// TIA Portal V17 export
// export: Created 2025-03-05T08:03:12.6134683Z, ExportSetting WithDefaults, DisplayName Totally Integrated Automation Portal, DisplayVersion V17 Update 8, DisplayName TIA Portal Openness, DisplayVersion V17 Update 8, DisplayName TIA Portal Version Control Interface, DisplayVersion V17, DisplayName SINAMICS Startdrive Advanced, DisplayVersion V17 SP2, DisplayName SINAMICS Startdrive G110M, G120, G120C, G120D, G120P, G115D, DisplayVersion V17 SP2, DisplayName SINAMICS Startdrive G130, G150, S120, S150, SINAMICS MV, S210, DisplayVersion V17 SP2, DisplayName STEP 7 Professional, DisplayVersion V17 Update 8, DisplayName SINUMERIK ONE STEP 7 Toolbox, DisplayVersion V17 Update 12, DisplayName SINUMERIK 840D sl STEP 7 Toolbox, DisplayVersion V17 Update 12, DisplayName STEP 7 Safety, DisplayVersion V17 Update 6, DisplayName WinCC Advanced, DisplayVersion V17 Update 8
FUNCTION "FC22500_HOPPER_SYSTEM_CONTROLS" : Void   // FC22500, LAD
TITLE = FC22500 HOPPER SYSTEM CONTROLS
{ S7_Optimized_Access := 'TRUE' }
VERSION : 0.1
// stored: AutoNumber false, IsIECCheckEnabled false, SetENOAutomatically false, UDAEnableTagReadback false
   VAR_TEMP
      RPM_INT_AUX : Word;
      RPM_REAL_AUX : Real;
   END_VAR
BEGIN

REGION Network 1: //////////UNIT 01 HOPERS CONTROLS//////////
END_REGION

REGION Network 2: CALL FB22501 TEMPERATURE JKT CONTROL UPPER HOPPER 1 UNIT 01
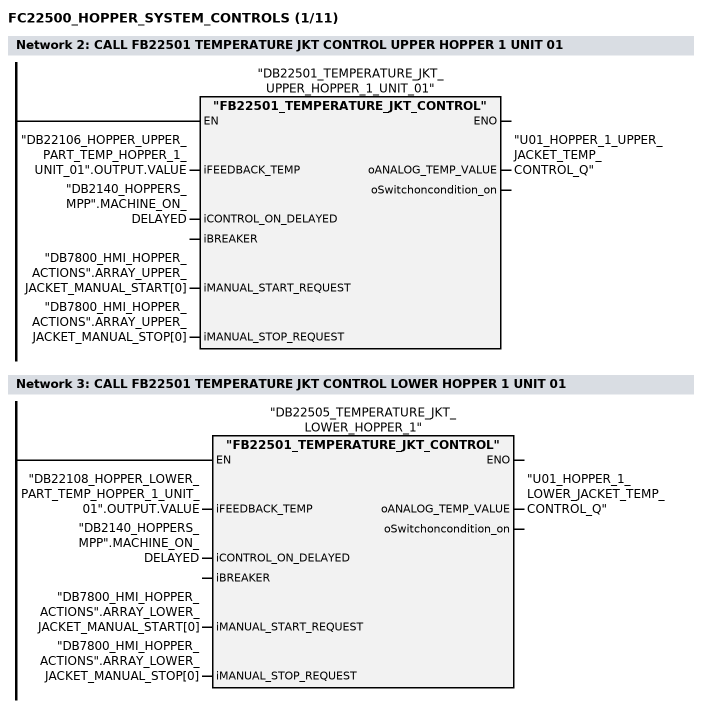
   RUNG wire#powerrail
      "DB22501_TEMPERATURE_JKT_UPPER_HOPPER_1_UNIT_01"(iFEEDBACK_TEMP := "DB22106_HOPPER_UPPER_PART_TEMP_HOPPER_1_UNIT_01".OUTPUT.VALUE, iCONTROL_ON_DELAYED := "DB2140_HOPPERS_MPP".MACHINE_ON_DELAYED, iBREAKER :=, iMANUAL_START_REQUEST := "DB7800_HMI_HOPPER_ACTIONS".ARRAY_UPPER_JACKET_MANUAL_START[0], iMANUAL_STOP_REQUEST := "DB7800_HMI_HOPPER_ACTIONS".ARRAY_UPPER_JACKET_MANUAL_STOP[0], oANALOG_TEMP_VALUE => "U01_HOPPER_1_UPPER_JACKET_TEMP_CONTROL_Q", oSwitchoncondition_on =>)
   END_RUNG
   // the same network as SCL:
   "DB22501_TEMPERATURE_JKT_UPPER_HOPPER_1_UNIT_01"(iFEEDBACK_TEMP := "DB22106_HOPPER_UPPER_PART_TEMP_HOPPER_1_UNIT_01".OUTPUT.VALUE,   // "FB22501_TEMPERATURE_JKT_CONTROL"
                           iCONTROL_ON_DELAYED := "DB2140_HOPPERS_MPP".MACHINE_ON_DELAYED,
                           iMANUAL_START_REQUEST := "DB7800_HMI_HOPPER_ACTIONS".ARRAY_UPPER_JACKET_MANUAL_START[0],
                           iMANUAL_STOP_REQUEST := "DB7800_HMI_HOPPER_ACTIONS".ARRAY_UPPER_JACKET_MANUAL_STOP[0],
                           oANALOG_TEMP_VALUE => "U01_HOPPER_1_UPPER_JACKET_TEMP_CONTROL_Q");
END_REGION

REGION Network 3: CALL FB22501 TEMPERATURE JKT CONTROL LOWER HOPPER 1 UNIT 01
   RUNG wire#powerrail
      "DB22505_TEMPERATURE_JKT_LOWER_HOPPER_1"(iFEEDBACK_TEMP := "DB22108_HOPPER_LOWER_PART_TEMP_HOPPER_1_UNIT_01".OUTPUT.VALUE, iCONTROL_ON_DELAYED := "DB2140_HOPPERS_MPP".MACHINE_ON_DELAYED, iBREAKER :=, iMANUAL_START_REQUEST := "DB7800_HMI_HOPPER_ACTIONS".ARRAY_LOWER_JACKET_MANUAL_START[0], iMANUAL_STOP_REQUEST := "DB7800_HMI_HOPPER_ACTIONS".ARRAY_LOWER_JACKET_MANUAL_STOP[0], oANALOG_TEMP_VALUE => "U01_HOPPER_1_LOWER_JACKET_TEMP_CONTROL_Q", oSwitchoncondition_on =>)
   END_RUNG
   // the same network as SCL:
   "DB22505_TEMPERATURE_JKT_LOWER_HOPPER_1"(iFEEDBACK_TEMP := "DB22108_HOPPER_LOWER_PART_TEMP_HOPPER_1_UNIT_01".OUTPUT.VALUE,   // "FB22501_TEMPERATURE_JKT_CONTROL"
                           iCONTROL_ON_DELAYED := "DB2140_HOPPERS_MPP".MACHINE_ON_DELAYED,
                           iMANUAL_START_REQUEST := "DB7800_HMI_HOPPER_ACTIONS".ARRAY_LOWER_JACKET_MANUAL_START[0],
                           iMANUAL_STOP_REQUEST := "DB7800_HMI_HOPPER_ACTIONS".ARRAY_LOWER_JACKET_MANUAL_STOP[0],
                           oANALOG_TEMP_VALUE => "U01_HOPPER_1_LOWER_JACKET_TEMP_CONTROL_Q");
END_REGION

REGION Network 4: CALL FB22502 MOTOR STIRRER CONTROL HOPPER 1 UNIT 01
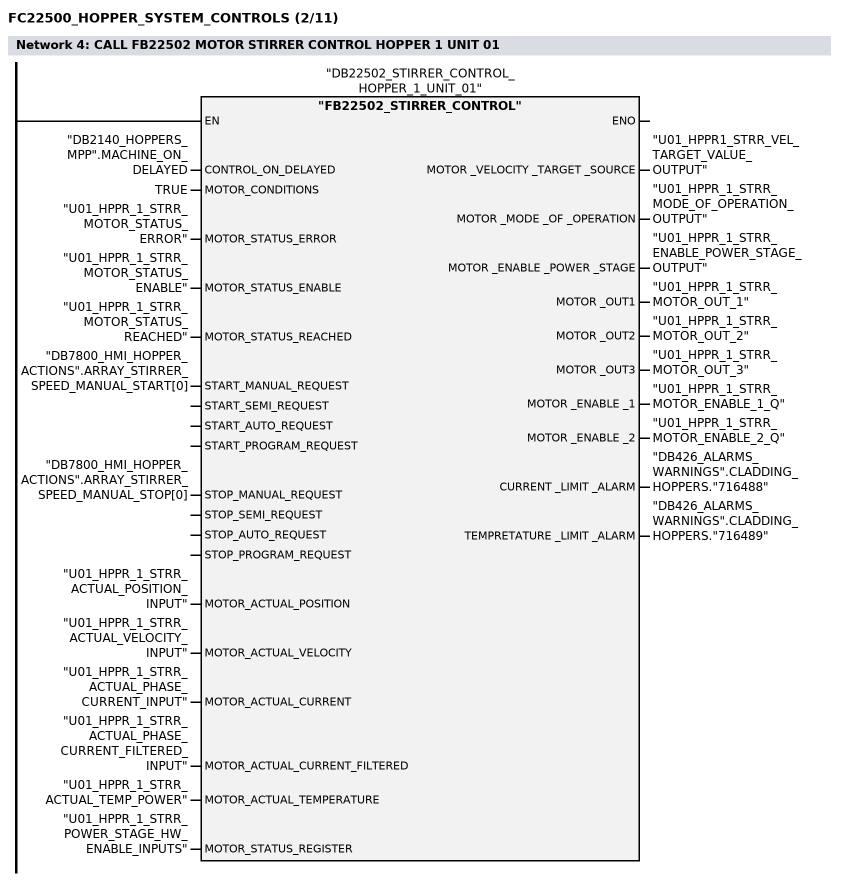
   RUNG wire#powerrail
      "DB22502_STIRRER_CONTROL_HOPPER_1_UNIT_01"(CONTROL_ON_DELAYED := "DB2140_HOPPERS_MPP".MACHINE_ON_DELAYED, MOTOR_CONDITIONS := TRUE, MOTOR_STATUS_ERROR := "U01_HPPR_1_STRR_MOTOR_STATUS_ERROR", MOTOR_STATUS_ENABLE := "U01_HPPR_1_STRR_MOTOR_STATUS_ENABLE", MOTOR_STATUS_REACHED := "U01_HPPR_1_STRR_MOTOR_STATUS_REACHED", START_MANUAL_REQUEST := "DB7800_HMI_HOPPER_ACTIONS".ARRAY_STIRRER_SPEED_MANUAL_START[0], START_SEMI_REQUEST :=, START_AUTO_REQUEST :=, START_PROGRAM_REQUEST :=, STOP_MANUAL_REQUEST := "DB7800_HMI_HOPPER_ACTIONS".ARRAY_STIRRER_SPEED_MANUAL_STOP[0], STOP_SEMI_REQUEST :=, STOP_AUTO_REQUEST :=, STOP_PROGRAM_REQUEST :=, MOTOR_ACTUAL_POSITION := "U01_HPPR_1_STRR_ACTUAL_POSITION_INPUT", MOTOR_ACTUAL_VELOCITY := "U01_HPPR_1_STRR_ACTUAL_VELOCITY_INPUT", MOTOR_ACTUAL_CURRENT := "U01_HPPR_1_STRR_ACTUAL_PHASE_CURRENT_INPUT", MOTOR_ACTUAL_CURRENT_FILTERED := "U01_HPPR_1_STRR_ACTUAL_PHASE_CURRENT_FILTERED_INPUT", MOTOR_ACTUAL_TEMPERATURE := "U01_HPPR_1_STRR_ACTUAL_TEMP_POWER", MOTOR_STATUS_REGISTER := "U01_HPPR_1_STRR_POWER_STAGE_HW_ENABLE_INPUTS", "MOTOR _VELOCITY _TARGET _SOURCE" => "U01_HPPR1_STRR_VEL_TARGET_VALUE_OUTPUT", "MOTOR _MODE _OF _OPERATION" => "U01_HPPR_1_STRR_MODE_OF_OPERATION_OUTPUT", "MOTOR _ENABLE _POWER _STAGE" => "U01_HPPR_1_STRR_ENABLE_POWER_STAGE_OUTPUT", "MOTOR _OUT1" => "U01_HPPR_1_STRR_MOTOR_OUT_1", "MOTOR _OUT2" => "U01_HPPR_1_STRR_MOTOR_OUT_2", "MOTOR _OUT3" => "U01_HPPR_1_STRR_MOTOR_OUT_3", "MOTOR _ENABLE _1" => "U01_HPPR_1_STRR_MOTOR_ENABLE_1_Q", "MOTOR _ENABLE _2" => "U01_HPPR_1_STRR_MOTOR_ENABLE_2_Q", "CURRENT _LIMIT _ALARM" => "DB426_ALARMS_WARNINGS".CLADDING_HOPPERS."716488", "TEMPRETATURE _LIMIT _ALARM" => "DB426_ALARMS_WARNINGS".CLADDING_HOPPERS."716489")
   END_RUNG
   // the same network as SCL:
   "DB22502_STIRRER_CONTROL_HOPPER_1_UNIT_01"(CONTROL_ON_DELAYED := "DB2140_HOPPERS_MPP".MACHINE_ON_DELAYED,   // "FB22502_STIRRER_CONTROL"
                           MOTOR_CONDITIONS := TRUE,
                           MOTOR_STATUS_ERROR := "U01_HPPR_1_STRR_MOTOR_STATUS_ERROR",
                           MOTOR_STATUS_ENABLE := "U01_HPPR_1_STRR_MOTOR_STATUS_ENABLE",
                           MOTOR_STATUS_REACHED := "U01_HPPR_1_STRR_MOTOR_STATUS_REACHED",
                           START_MANUAL_REQUEST := "DB7800_HMI_HOPPER_ACTIONS".ARRAY_STIRRER_SPEED_MANUAL_START[0],
                           STOP_MANUAL_REQUEST := "DB7800_HMI_HOPPER_ACTIONS".ARRAY_STIRRER_SPEED_MANUAL_STOP[0],
                           MOTOR_ACTUAL_POSITION := "U01_HPPR_1_STRR_ACTUAL_POSITION_INPUT",
                           MOTOR_ACTUAL_VELOCITY := "U01_HPPR_1_STRR_ACTUAL_VELOCITY_INPUT",
                           MOTOR_ACTUAL_CURRENT := "U01_HPPR_1_STRR_ACTUAL_PHASE_CURRENT_INPUT",
                           MOTOR_ACTUAL_CURRENT_FILTERED := "U01_HPPR_1_STRR_ACTUAL_PHASE_CURRENT_FILTERED_INPUT",
                           MOTOR_ACTUAL_TEMPERATURE := "U01_HPPR_1_STRR_ACTUAL_TEMP_POWER",
                           MOTOR_STATUS_REGISTER := "U01_HPPR_1_STRR_POWER_STAGE_HW_ENABLE_INPUTS",
                           "MOTOR _VELOCITY _TARGET _SOURCE" => "U01_HPPR1_STRR_VEL_TARGET_VALUE_OUTPUT",
                           "MOTOR _MODE _OF _OPERATION" => "U01_HPPR_1_STRR_MODE_OF_OPERATION_OUTPUT",
                           "MOTOR _ENABLE _POWER _STAGE" => "U01_HPPR_1_STRR_ENABLE_POWER_STAGE_OUTPUT",
                           "MOTOR _OUT1" => "U01_HPPR_1_STRR_MOTOR_OUT_1",
                           "MOTOR _OUT2" => "U01_HPPR_1_STRR_MOTOR_OUT_2",
                           "MOTOR _OUT3" => "U01_HPPR_1_STRR_MOTOR_OUT_3",
                           "MOTOR _ENABLE _1" => "U01_HPPR_1_STRR_MOTOR_ENABLE_1_Q",
                           "MOTOR _ENABLE _2" => "U01_HPPR_1_STRR_MOTOR_ENABLE_2_Q",
                           "CURRENT _LIMIT _ALARM" => "DB426_ALARMS_WARNINGS".CLADDING_HOPPERS."716488",
                           "TEMPRETATURE _LIMIT _ALARM" => "DB426_ALARMS_WARNINGS".CLADDING_HOPPERS."716489");
END_REGION

REGION Network 5: CALL FB22503 HOPPER COVER PRESSURE CONTROL HOPPER 1 UNIT 01
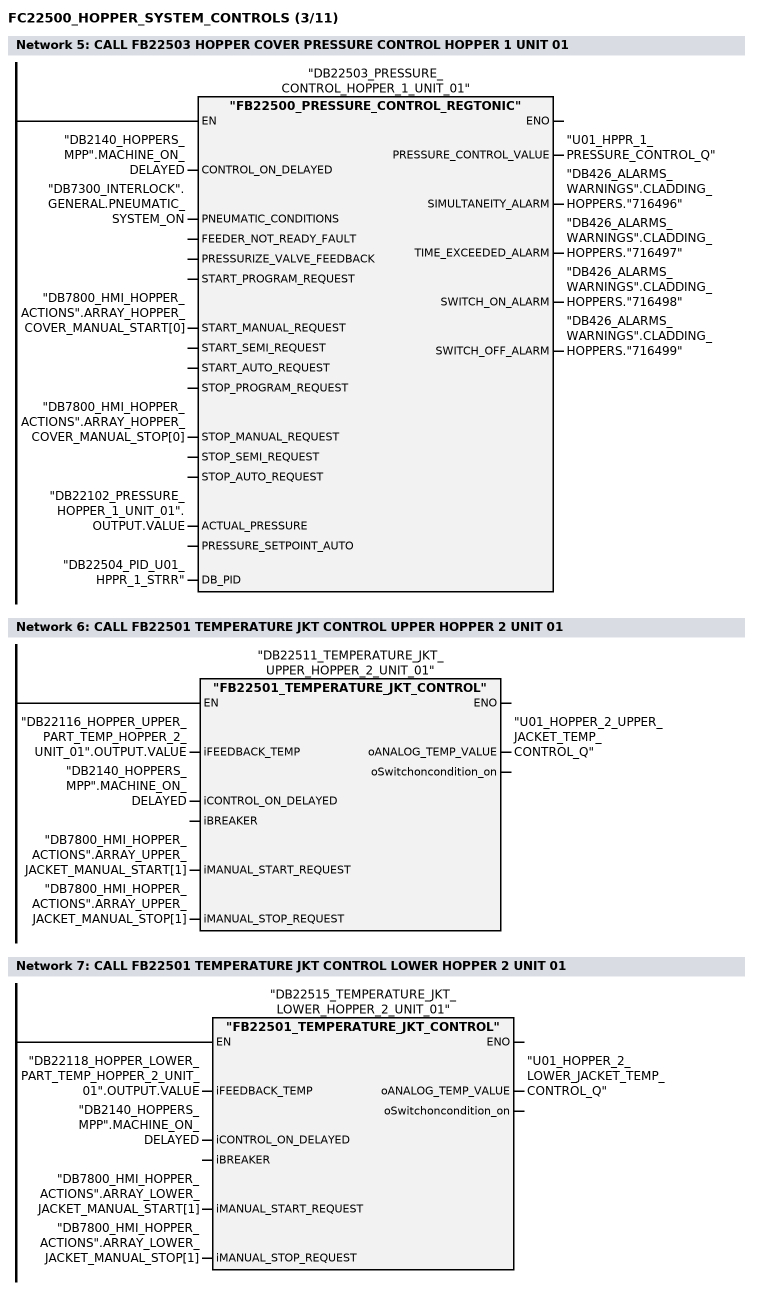
   RUNG wire#powerrail
      "DB22503_PRESSURE_CONTROL_HOPPER_1_UNIT_01"(CONTROL_ON_DELAYED := "DB2140_HOPPERS_MPP".MACHINE_ON_DELAYED, PNEUMATIC_CONDITIONS := "DB7300_INTERLOCK".GENERAL.PNEUMATIC_SYSTEM_ON, FEEDER_NOT_READY_FAULT :=, PRESSURIZE_VALVE_FEEDBACK :=, START_PROGRAM_REQUEST :=, START_MANUAL_REQUEST := "DB7800_HMI_HOPPER_ACTIONS".ARRAY_HOPPER_COVER_MANUAL_START[0], START_SEMI_REQUEST :=, START_AUTO_REQUEST :=, STOP_PROGRAM_REQUEST :=, STOP_MANUAL_REQUEST := "DB7800_HMI_HOPPER_ACTIONS".ARRAY_HOPPER_COVER_MANUAL_STOP[0], STOP_SEMI_REQUEST :=, STOP_AUTO_REQUEST :=, ACTUAL_PRESSURE := "DB22102_PRESSURE_HOPPER_1_UNIT_01".OUTPUT.VALUE, PRESSURE_SETPOINT_AUTO :=, DB_PID := "DB22504_PID_U01_HPPR_1_STRR", PRESSURE_CONTROL_VALUE => "U01_HPPR_1_PRESSURE_CONTROL_Q", SIMULTANEITY_ALARM => "DB426_ALARMS_WARNINGS".CLADDING_HOPPERS."716496", TIME_EXCEEDED_ALARM => "DB426_ALARMS_WARNINGS".CLADDING_HOPPERS."716497", SWITCH_ON_ALARM => "DB426_ALARMS_WARNINGS".CLADDING_HOPPERS."716498", SWITCH_OFF_ALARM => "DB426_ALARMS_WARNINGS".CLADDING_HOPPERS."716499")
   END_RUNG
   // the same network as SCL:
   "DB22503_PRESSURE_CONTROL_HOPPER_1_UNIT_01"(CONTROL_ON_DELAYED := "DB2140_HOPPERS_MPP".MACHINE_ON_DELAYED,   // "FB22500_PRESSURE_CONTROL_REGTONIC"
                           PNEUMATIC_CONDITIONS := "DB7300_INTERLOCK".GENERAL.PNEUMATIC_SYSTEM_ON,
                           START_MANUAL_REQUEST := "DB7800_HMI_HOPPER_ACTIONS".ARRAY_HOPPER_COVER_MANUAL_START[0],
                           STOP_MANUAL_REQUEST := "DB7800_HMI_HOPPER_ACTIONS".ARRAY_HOPPER_COVER_MANUAL_STOP[0],
                           ACTUAL_PRESSURE := "DB22102_PRESSURE_HOPPER_1_UNIT_01".OUTPUT.VALUE,
                           DB_PID := "DB22504_PID_U01_HPPR_1_STRR",
                           PRESSURE_CONTROL_VALUE => "U01_HPPR_1_PRESSURE_CONTROL_Q",
                           SIMULTANEITY_ALARM => "DB426_ALARMS_WARNINGS".CLADDING_HOPPERS."716496",
                           TIME_EXCEEDED_ALARM => "DB426_ALARMS_WARNINGS".CLADDING_HOPPERS."716497",
                           SWITCH_ON_ALARM => "DB426_ALARMS_WARNINGS".CLADDING_HOPPERS."716498",
                           SWITCH_OFF_ALARM => "DB426_ALARMS_WARNINGS".CLADDING_HOPPERS."716499");
END_REGION

REGION Network 6: CALL FB22501 TEMPERATURE JKT CONTROL UPPER HOPPER 2 UNIT 01
   RUNG wire#powerrail
      "DB22511_TEMPERATURE_JKT_UPPER_HOPPER_2_UNIT_01"(iFEEDBACK_TEMP := "DB22116_HOPPER_UPPER_PART_TEMP_HOPPER_2_UNIT_01".OUTPUT.VALUE, iCONTROL_ON_DELAYED := "DB2140_HOPPERS_MPP".MACHINE_ON_DELAYED, iBREAKER :=, iMANUAL_START_REQUEST := "DB7800_HMI_HOPPER_ACTIONS".ARRAY_UPPER_JACKET_MANUAL_START[1], iMANUAL_STOP_REQUEST := "DB7800_HMI_HOPPER_ACTIONS".ARRAY_UPPER_JACKET_MANUAL_STOP[1], oANALOG_TEMP_VALUE => "U01_HOPPER_2_UPPER_JACKET_TEMP_CONTROL_Q", oSwitchoncondition_on =>)
   END_RUNG
   // the same network as SCL:
   "DB22511_TEMPERATURE_JKT_UPPER_HOPPER_2_UNIT_01"(iFEEDBACK_TEMP := "DB22116_HOPPER_UPPER_PART_TEMP_HOPPER_2_UNIT_01".OUTPUT.VALUE,   // "FB22501_TEMPERATURE_JKT_CONTROL"
                           iCONTROL_ON_DELAYED := "DB2140_HOPPERS_MPP".MACHINE_ON_DELAYED,
                           iMANUAL_START_REQUEST := "DB7800_HMI_HOPPER_ACTIONS".ARRAY_UPPER_JACKET_MANUAL_START[1],
                           iMANUAL_STOP_REQUEST := "DB7800_HMI_HOPPER_ACTIONS".ARRAY_UPPER_JACKET_MANUAL_STOP[1],
                           oANALOG_TEMP_VALUE => "U01_HOPPER_2_UPPER_JACKET_TEMP_CONTROL_Q");
END_REGION

REGION Network 7: CALL FB22501 TEMPERATURE JKT CONTROL LOWER HOPPER 2 UNIT 01
   RUNG wire#powerrail
      "DB22515_TEMPERATURE_JKT_LOWER_HOPPER_2_UNIT_01"(iFEEDBACK_TEMP := "DB22118_HOPPER_LOWER_PART_TEMP_HOPPER_2_UNIT_01".OUTPUT.VALUE, iCONTROL_ON_DELAYED := "DB2140_HOPPERS_MPP".MACHINE_ON_DELAYED, iBREAKER :=, iMANUAL_START_REQUEST := "DB7800_HMI_HOPPER_ACTIONS".ARRAY_LOWER_JACKET_MANUAL_START[1], iMANUAL_STOP_REQUEST := "DB7800_HMI_HOPPER_ACTIONS".ARRAY_LOWER_JACKET_MANUAL_STOP[1], oANALOG_TEMP_VALUE => "U01_HOPPER_2_LOWER_JACKET_TEMP_CONTROL_Q", oSwitchoncondition_on =>)
   END_RUNG
   // the same network as SCL:
   "DB22515_TEMPERATURE_JKT_LOWER_HOPPER_2_UNIT_01"(iFEEDBACK_TEMP := "DB22118_HOPPER_LOWER_PART_TEMP_HOPPER_2_UNIT_01".OUTPUT.VALUE,   // "FB22501_TEMPERATURE_JKT_CONTROL"
                           iCONTROL_ON_DELAYED := "DB2140_HOPPERS_MPP".MACHINE_ON_DELAYED,
                           iMANUAL_START_REQUEST := "DB7800_HMI_HOPPER_ACTIONS".ARRAY_LOWER_JACKET_MANUAL_START[1],
                           iMANUAL_STOP_REQUEST := "DB7800_HMI_HOPPER_ACTIONS".ARRAY_LOWER_JACKET_MANUAL_STOP[1],
                           oANALOG_TEMP_VALUE => "U01_HOPPER_2_LOWER_JACKET_TEMP_CONTROL_Q");
END_REGION

REGION Network 8: CALL FB22502 MOTOR STIRRER CONTROL HOPPER 2 UNIT 01
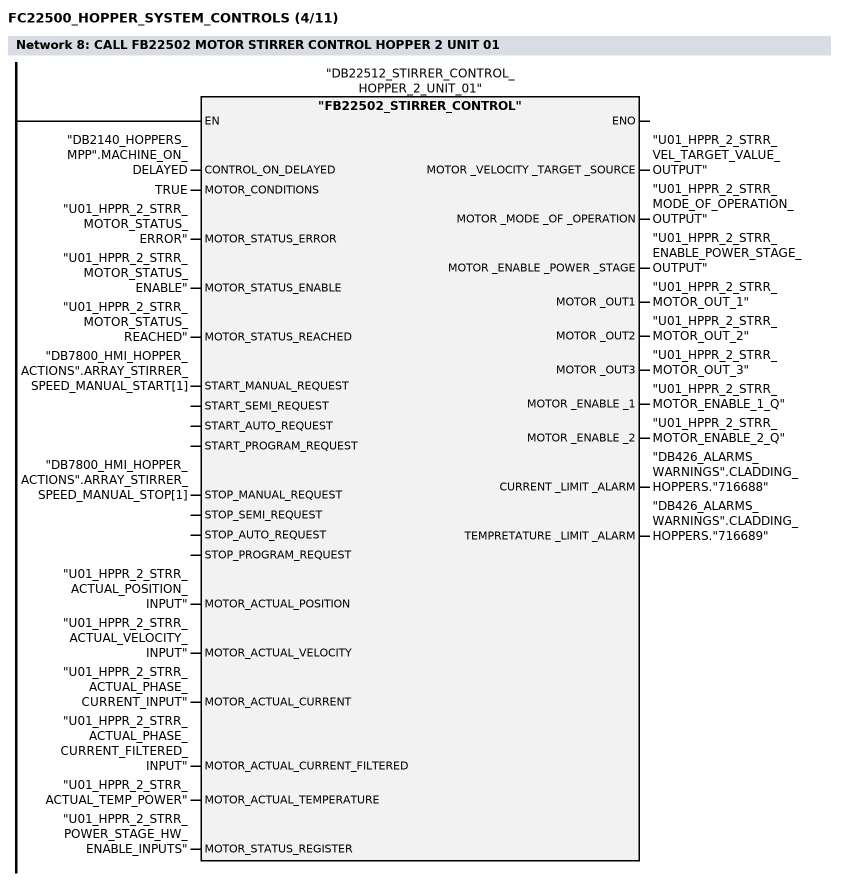
   RUNG wire#powerrail
      "DB22512_STIRRER_CONTROL_HOPPER_2_UNIT_01"(CONTROL_ON_DELAYED := "DB2140_HOPPERS_MPP".MACHINE_ON_DELAYED, MOTOR_CONDITIONS := TRUE, MOTOR_STATUS_ERROR := "U01_HPPR_2_STRR_MOTOR_STATUS_ERROR", MOTOR_STATUS_ENABLE := "U01_HPPR_2_STRR_MOTOR_STATUS_ENABLE", MOTOR_STATUS_REACHED := "U01_HPPR_2_STRR_MOTOR_STATUS_REACHED", START_MANUAL_REQUEST := "DB7800_HMI_HOPPER_ACTIONS".ARRAY_STIRRER_SPEED_MANUAL_START[1], START_SEMI_REQUEST :=, START_AUTO_REQUEST :=, START_PROGRAM_REQUEST :=, STOP_MANUAL_REQUEST := "DB7800_HMI_HOPPER_ACTIONS".ARRAY_STIRRER_SPEED_MANUAL_STOP[1], STOP_SEMI_REQUEST :=, STOP_AUTO_REQUEST :=, STOP_PROGRAM_REQUEST :=, MOTOR_ACTUAL_POSITION := "U01_HPPR_2_STRR_ACTUAL_POSITION_INPUT", MOTOR_ACTUAL_VELOCITY := "U01_HPPR_2_STRR_ACTUAL_VELOCITY_INPUT", MOTOR_ACTUAL_CURRENT := "U01_HPPR_2_STRR_ACTUAL_PHASE_CURRENT_INPUT", MOTOR_ACTUAL_CURRENT_FILTERED := "U01_HPPR_2_STRR_ACTUAL_PHASE_CURRENT_FILTERED_INPUT", MOTOR_ACTUAL_TEMPERATURE := "U01_HPPR_2_STRR_ACTUAL_TEMP_POWER", MOTOR_STATUS_REGISTER := "U01_HPPR_2_STRR_POWER_STAGE_HW_ENABLE_INPUTS", "MOTOR _VELOCITY _TARGET _SOURCE" => "U01_HPPR_2_STRR_VEL_TARGET_VALUE_OUTPUT", "MOTOR _MODE _OF _OPERATION" => "U01_HPPR_2_STRR_MODE_OF_OPERATION_OUTPUT", "MOTOR _ENABLE _POWER _STAGE" => "U01_HPPR_2_STRR_ENABLE_POWER_STAGE_OUTPUT", "MOTOR _OUT1" => "U01_HPPR_2_STRR_MOTOR_OUT_1", "MOTOR _OUT2" => "U01_HPPR_2_STRR_MOTOR_OUT_2", "MOTOR _OUT3" => "U01_HPPR_2_STRR_MOTOR_OUT_3", "MOTOR _ENABLE _1" => "U01_HPPR_2_STRR_MOTOR_ENABLE_1_Q", "MOTOR _ENABLE _2" => "U01_HPPR_2_STRR_MOTOR_ENABLE_2_Q", "CURRENT _LIMIT _ALARM" => "DB426_ALARMS_WARNINGS".CLADDING_HOPPERS."716688", "TEMPRETATURE _LIMIT _ALARM" => "DB426_ALARMS_WARNINGS".CLADDING_HOPPERS."716689")
   END_RUNG
   // the same network as SCL:
   "DB22512_STIRRER_CONTROL_HOPPER_2_UNIT_01"(CONTROL_ON_DELAYED := "DB2140_HOPPERS_MPP".MACHINE_ON_DELAYED,   // "FB22502_STIRRER_CONTROL"
                           MOTOR_CONDITIONS := TRUE,
                           MOTOR_STATUS_ERROR := "U01_HPPR_2_STRR_MOTOR_STATUS_ERROR",
                           MOTOR_STATUS_ENABLE := "U01_HPPR_2_STRR_MOTOR_STATUS_ENABLE",
                           MOTOR_STATUS_REACHED := "U01_HPPR_2_STRR_MOTOR_STATUS_REACHED",
                           START_MANUAL_REQUEST := "DB7800_HMI_HOPPER_ACTIONS".ARRAY_STIRRER_SPEED_MANUAL_START[1],
                           STOP_MANUAL_REQUEST := "DB7800_HMI_HOPPER_ACTIONS".ARRAY_STIRRER_SPEED_MANUAL_STOP[1],
                           MOTOR_ACTUAL_POSITION := "U01_HPPR_2_STRR_ACTUAL_POSITION_INPUT",
                           MOTOR_ACTUAL_VELOCITY := "U01_HPPR_2_STRR_ACTUAL_VELOCITY_INPUT",
                           MOTOR_ACTUAL_CURRENT := "U01_HPPR_2_STRR_ACTUAL_PHASE_CURRENT_INPUT",
                           MOTOR_ACTUAL_CURRENT_FILTERED := "U01_HPPR_2_STRR_ACTUAL_PHASE_CURRENT_FILTERED_INPUT",
                           MOTOR_ACTUAL_TEMPERATURE := "U01_HPPR_2_STRR_ACTUAL_TEMP_POWER",
                           MOTOR_STATUS_REGISTER := "U01_HPPR_2_STRR_POWER_STAGE_HW_ENABLE_INPUTS",
                           "MOTOR _VELOCITY _TARGET _SOURCE" => "U01_HPPR_2_STRR_VEL_TARGET_VALUE_OUTPUT",
                           "MOTOR _MODE _OF _OPERATION" => "U01_HPPR_2_STRR_MODE_OF_OPERATION_OUTPUT",
                           "MOTOR _ENABLE _POWER _STAGE" => "U01_HPPR_2_STRR_ENABLE_POWER_STAGE_OUTPUT",
                           "MOTOR _OUT1" => "U01_HPPR_2_STRR_MOTOR_OUT_1",
                           "MOTOR _OUT2" => "U01_HPPR_2_STRR_MOTOR_OUT_2",
                           "MOTOR _OUT3" => "U01_HPPR_2_STRR_MOTOR_OUT_3",
                           "MOTOR _ENABLE _1" => "U01_HPPR_2_STRR_MOTOR_ENABLE_1_Q",
                           "MOTOR _ENABLE _2" => "U01_HPPR_2_STRR_MOTOR_ENABLE_2_Q",
                           "CURRENT _LIMIT _ALARM" => "DB426_ALARMS_WARNINGS".CLADDING_HOPPERS."716688",
                           "TEMPRETATURE _LIMIT _ALARM" => "DB426_ALARMS_WARNINGS".CLADDING_HOPPERS."716689");
END_REGION

REGION Network 9: CALL FB22503 HOPPER PRESSURE CONTROL HOPPER 2 UNIT 01
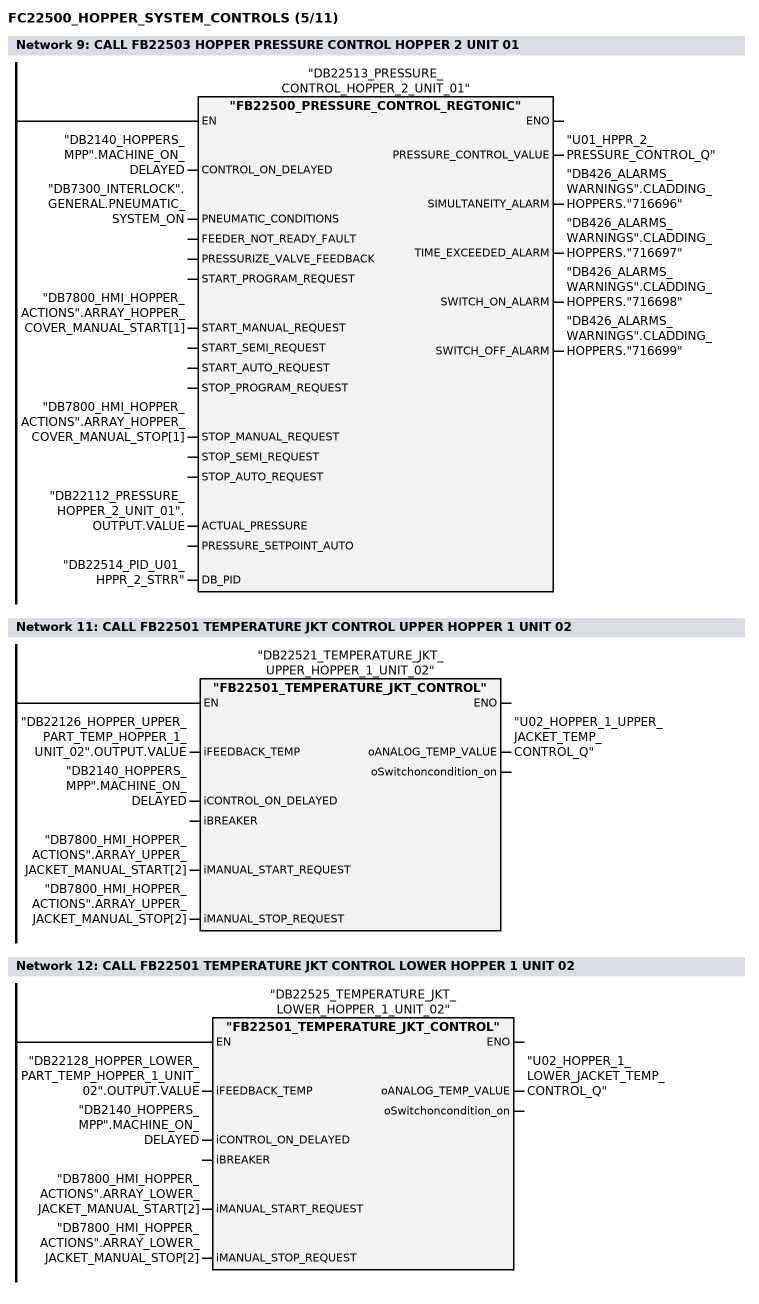
   RUNG wire#powerrail
      "DB22513_PRESSURE_CONTROL_HOPPER_2_UNIT_01"(CONTROL_ON_DELAYED := "DB2140_HOPPERS_MPP".MACHINE_ON_DELAYED, PNEUMATIC_CONDITIONS := "DB7300_INTERLOCK".GENERAL.PNEUMATIC_SYSTEM_ON, FEEDER_NOT_READY_FAULT :=, PRESSURIZE_VALVE_FEEDBACK :=, START_PROGRAM_REQUEST :=, START_MANUAL_REQUEST := "DB7800_HMI_HOPPER_ACTIONS".ARRAY_HOPPER_COVER_MANUAL_START[1], START_SEMI_REQUEST :=, START_AUTO_REQUEST :=, STOP_PROGRAM_REQUEST :=, STOP_MANUAL_REQUEST := "DB7800_HMI_HOPPER_ACTIONS".ARRAY_HOPPER_COVER_MANUAL_STOP[1], STOP_SEMI_REQUEST :=, STOP_AUTO_REQUEST :=, ACTUAL_PRESSURE := "DB22112_PRESSURE_HOPPER_2_UNIT_01".OUTPUT.VALUE, PRESSURE_SETPOINT_AUTO :=, DB_PID := "DB22514_PID_U01_HPPR_2_STRR", PRESSURE_CONTROL_VALUE => "U01_HPPR_2_PRESSURE_CONTROL_Q", SIMULTANEITY_ALARM => "DB426_ALARMS_WARNINGS".CLADDING_HOPPERS."716696", TIME_EXCEEDED_ALARM => "DB426_ALARMS_WARNINGS".CLADDING_HOPPERS."716697", SWITCH_ON_ALARM => "DB426_ALARMS_WARNINGS".CLADDING_HOPPERS."716698", SWITCH_OFF_ALARM => "DB426_ALARMS_WARNINGS".CLADDING_HOPPERS."716699")
   END_RUNG
   // the same network as SCL:
   "DB22513_PRESSURE_CONTROL_HOPPER_2_UNIT_01"(CONTROL_ON_DELAYED := "DB2140_HOPPERS_MPP".MACHINE_ON_DELAYED,   // "FB22500_PRESSURE_CONTROL_REGTONIC"
                           PNEUMATIC_CONDITIONS := "DB7300_INTERLOCK".GENERAL.PNEUMATIC_SYSTEM_ON,
                           START_MANUAL_REQUEST := "DB7800_HMI_HOPPER_ACTIONS".ARRAY_HOPPER_COVER_MANUAL_START[1],
                           STOP_MANUAL_REQUEST := "DB7800_HMI_HOPPER_ACTIONS".ARRAY_HOPPER_COVER_MANUAL_STOP[1],
                           ACTUAL_PRESSURE := "DB22112_PRESSURE_HOPPER_2_UNIT_01".OUTPUT.VALUE,
                           DB_PID := "DB22514_PID_U01_HPPR_2_STRR",
                           PRESSURE_CONTROL_VALUE => "U01_HPPR_2_PRESSURE_CONTROL_Q",
                           SIMULTANEITY_ALARM => "DB426_ALARMS_WARNINGS".CLADDING_HOPPERS."716696",
                           TIME_EXCEEDED_ALARM => "DB426_ALARMS_WARNINGS".CLADDING_HOPPERS."716697",
                           SWITCH_ON_ALARM => "DB426_ALARMS_WARNINGS".CLADDING_HOPPERS."716698",
                           SWITCH_OFF_ALARM => "DB426_ALARMS_WARNINGS".CLADDING_HOPPERS."716699");
END_REGION

REGION Network 10: //////////UNIT 02 HOPERS CONTROLS//////////
END_REGION

REGION Network 11: CALL FB22501 TEMPERATURE JKT CONTROL UPPER HOPPER 1 UNIT 02
   RUNG wire#powerrail
      "DB22521_TEMPERATURE_JKT_UPPER_HOPPER_1_UNIT_02"(iFEEDBACK_TEMP := "DB22126_HOPPER_UPPER_PART_TEMP_HOPPER_1_UNIT_02".OUTPUT.VALUE, iCONTROL_ON_DELAYED := "DB2140_HOPPERS_MPP".MACHINE_ON_DELAYED, iBREAKER :=, iMANUAL_START_REQUEST := "DB7800_HMI_HOPPER_ACTIONS".ARRAY_UPPER_JACKET_MANUAL_START[2], iMANUAL_STOP_REQUEST := "DB7800_HMI_HOPPER_ACTIONS".ARRAY_UPPER_JACKET_MANUAL_STOP[2], oANALOG_TEMP_VALUE => "U02_HOPPER_1_UPPER_JACKET_TEMP_CONTROL_Q", oSwitchoncondition_on =>)
   END_RUNG
   // the same network as SCL:
   "DB22521_TEMPERATURE_JKT_UPPER_HOPPER_1_UNIT_02"(iFEEDBACK_TEMP := "DB22126_HOPPER_UPPER_PART_TEMP_HOPPER_1_UNIT_02".OUTPUT.VALUE,   // "FB22501_TEMPERATURE_JKT_CONTROL"
                           iCONTROL_ON_DELAYED := "DB2140_HOPPERS_MPP".MACHINE_ON_DELAYED,
                           iMANUAL_START_REQUEST := "DB7800_HMI_HOPPER_ACTIONS".ARRAY_UPPER_JACKET_MANUAL_START[2],
                           iMANUAL_STOP_REQUEST := "DB7800_HMI_HOPPER_ACTIONS".ARRAY_UPPER_JACKET_MANUAL_STOP[2],
                           oANALOG_TEMP_VALUE => "U02_HOPPER_1_UPPER_JACKET_TEMP_CONTROL_Q");
END_REGION

REGION Network 12: CALL FB22501 TEMPERATURE JKT CONTROL LOWER HOPPER 1 UNIT 02
   RUNG wire#powerrail
      "DB22525_TEMPERATURE_JKT_LOWER_HOPPER_1_UNIT_02"(iFEEDBACK_TEMP := "DB22128_HOPPER_LOWER_PART_TEMP_HOPPER_1_UNIT_02".OUTPUT.VALUE, iCONTROL_ON_DELAYED := "DB2140_HOPPERS_MPP".MACHINE_ON_DELAYED, iBREAKER :=, iMANUAL_START_REQUEST := "DB7800_HMI_HOPPER_ACTIONS".ARRAY_LOWER_JACKET_MANUAL_START[2], iMANUAL_STOP_REQUEST := "DB7800_HMI_HOPPER_ACTIONS".ARRAY_LOWER_JACKET_MANUAL_STOP[2], oANALOG_TEMP_VALUE => "U02_HOPPER_1_LOWER_JACKET_TEMP_CONTROL_Q", oSwitchoncondition_on =>)
   END_RUNG
   // the same network as SCL:
   "DB22525_TEMPERATURE_JKT_LOWER_HOPPER_1_UNIT_02"(iFEEDBACK_TEMP := "DB22128_HOPPER_LOWER_PART_TEMP_HOPPER_1_UNIT_02".OUTPUT.VALUE,   // "FB22501_TEMPERATURE_JKT_CONTROL"
                           iCONTROL_ON_DELAYED := "DB2140_HOPPERS_MPP".MACHINE_ON_DELAYED,
                           iMANUAL_START_REQUEST := "DB7800_HMI_HOPPER_ACTIONS".ARRAY_LOWER_JACKET_MANUAL_START[2],
                           iMANUAL_STOP_REQUEST := "DB7800_HMI_HOPPER_ACTIONS".ARRAY_LOWER_JACKET_MANUAL_STOP[2],
                           oANALOG_TEMP_VALUE => "U02_HOPPER_1_LOWER_JACKET_TEMP_CONTROL_Q");
END_REGION

REGION Network 13: CALL FB22502 MOTOR STIRRER CONTROL HOPPER 1 UNIT 02
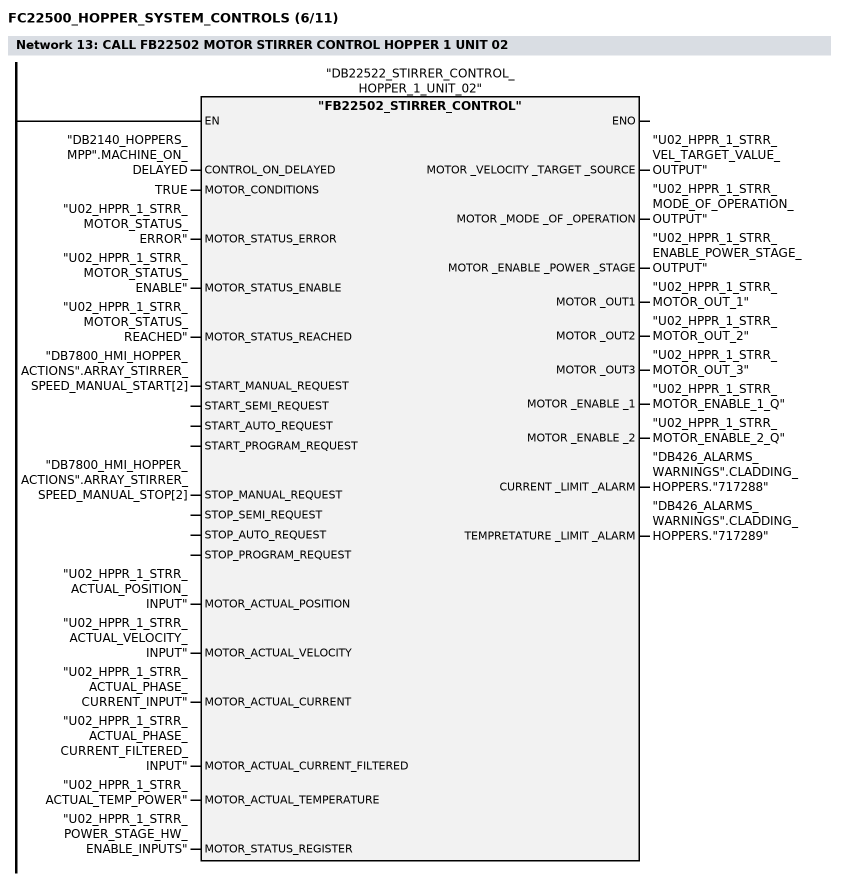
   RUNG wire#powerrail
      "DB22522_STIRRER_CONTROL_HOPPER_1_UNIT_02"(CONTROL_ON_DELAYED := "DB2140_HOPPERS_MPP".MACHINE_ON_DELAYED, MOTOR_CONDITIONS := TRUE, MOTOR_STATUS_ERROR := "U02_HPPR_1_STRR_MOTOR_STATUS_ERROR", MOTOR_STATUS_ENABLE := "U02_HPPR_1_STRR_MOTOR_STATUS_ENABLE", MOTOR_STATUS_REACHED := "U02_HPPR_1_STRR_MOTOR_STATUS_REACHED", START_MANUAL_REQUEST := "DB7800_HMI_HOPPER_ACTIONS".ARRAY_STIRRER_SPEED_MANUAL_START[2], START_SEMI_REQUEST :=, START_AUTO_REQUEST :=, START_PROGRAM_REQUEST :=, STOP_MANUAL_REQUEST := "DB7800_HMI_HOPPER_ACTIONS".ARRAY_STIRRER_SPEED_MANUAL_STOP[2], STOP_SEMI_REQUEST :=, STOP_AUTO_REQUEST :=, STOP_PROGRAM_REQUEST :=, MOTOR_ACTUAL_POSITION := "U02_HPPR_1_STRR_ACTUAL_POSITION_INPUT", MOTOR_ACTUAL_VELOCITY := "U02_HPPR_1_STRR_ACTUAL_VELOCITY_INPUT", MOTOR_ACTUAL_CURRENT := "U02_HPPR_1_STRR_ACTUAL_PHASE_CURRENT_INPUT", MOTOR_ACTUAL_CURRENT_FILTERED := "U02_HPPR_1_STRR_ACTUAL_PHASE_CURRENT_FILTERED_INPUT", MOTOR_ACTUAL_TEMPERATURE := "U02_HPPR_1_STRR_ACTUAL_TEMP_POWER", MOTOR_STATUS_REGISTER := "U02_HPPR_1_STRR_POWER_STAGE_HW_ENABLE_INPUTS", "MOTOR _VELOCITY _TARGET _SOURCE" => "U02_HPPR_1_STRR_VEL_TARGET_VALUE_OUTPUT", "MOTOR _MODE _OF _OPERATION" => "U02_HPPR_1_STRR_MODE_OF_OPERATION_OUTPUT", "MOTOR _ENABLE _POWER _STAGE" => "U02_HPPR_1_STRR_ENABLE_POWER_STAGE_OUTPUT", "MOTOR _OUT1" => "U02_HPPR_1_STRR_MOTOR_OUT_1", "MOTOR _OUT2" => "U02_HPPR_1_STRR_MOTOR_OUT_2", "MOTOR _OUT3" => "U02_HPPR_1_STRR_MOTOR_OUT_3", "MOTOR _ENABLE _1" => "U02_HPPR_1_STRR_MOTOR_ENABLE_1_Q", "MOTOR _ENABLE _2" => "U02_HPPR_1_STRR_MOTOR_ENABLE_2_Q", "CURRENT _LIMIT _ALARM" => "DB426_ALARMS_WARNINGS".CLADDING_HOPPERS."717288", "TEMPRETATURE _LIMIT _ALARM" => "DB426_ALARMS_WARNINGS".CLADDING_HOPPERS."717289")
   END_RUNG
   // the same network as SCL:
   "DB22522_STIRRER_CONTROL_HOPPER_1_UNIT_02"(CONTROL_ON_DELAYED := "DB2140_HOPPERS_MPP".MACHINE_ON_DELAYED,   // "FB22502_STIRRER_CONTROL"
                           MOTOR_CONDITIONS := TRUE,
                           MOTOR_STATUS_ERROR := "U02_HPPR_1_STRR_MOTOR_STATUS_ERROR",
                           MOTOR_STATUS_ENABLE := "U02_HPPR_1_STRR_MOTOR_STATUS_ENABLE",
                           MOTOR_STATUS_REACHED := "U02_HPPR_1_STRR_MOTOR_STATUS_REACHED",
                           START_MANUAL_REQUEST := "DB7800_HMI_HOPPER_ACTIONS".ARRAY_STIRRER_SPEED_MANUAL_START[2],
                           STOP_MANUAL_REQUEST := "DB7800_HMI_HOPPER_ACTIONS".ARRAY_STIRRER_SPEED_MANUAL_STOP[2],
                           MOTOR_ACTUAL_POSITION := "U02_HPPR_1_STRR_ACTUAL_POSITION_INPUT",
                           MOTOR_ACTUAL_VELOCITY := "U02_HPPR_1_STRR_ACTUAL_VELOCITY_INPUT",
                           MOTOR_ACTUAL_CURRENT := "U02_HPPR_1_STRR_ACTUAL_PHASE_CURRENT_INPUT",
                           MOTOR_ACTUAL_CURRENT_FILTERED := "U02_HPPR_1_STRR_ACTUAL_PHASE_CURRENT_FILTERED_INPUT",
                           MOTOR_ACTUAL_TEMPERATURE := "U02_HPPR_1_STRR_ACTUAL_TEMP_POWER",
                           MOTOR_STATUS_REGISTER := "U02_HPPR_1_STRR_POWER_STAGE_HW_ENABLE_INPUTS",
                           "MOTOR _VELOCITY _TARGET _SOURCE" => "U02_HPPR_1_STRR_VEL_TARGET_VALUE_OUTPUT",
                           "MOTOR _MODE _OF _OPERATION" => "U02_HPPR_1_STRR_MODE_OF_OPERATION_OUTPUT",
                           "MOTOR _ENABLE _POWER _STAGE" => "U02_HPPR_1_STRR_ENABLE_POWER_STAGE_OUTPUT",
                           "MOTOR _OUT1" => "U02_HPPR_1_STRR_MOTOR_OUT_1",
                           "MOTOR _OUT2" => "U02_HPPR_1_STRR_MOTOR_OUT_2",
                           "MOTOR _OUT3" => "U02_HPPR_1_STRR_MOTOR_OUT_3",
                           "MOTOR _ENABLE _1" => "U02_HPPR_1_STRR_MOTOR_ENABLE_1_Q",
                           "MOTOR _ENABLE _2" => "U02_HPPR_1_STRR_MOTOR_ENABLE_2_Q",
                           "CURRENT _LIMIT _ALARM" => "DB426_ALARMS_WARNINGS".CLADDING_HOPPERS."717288",
                           "TEMPRETATURE _LIMIT _ALARM" => "DB426_ALARMS_WARNINGS".CLADDING_HOPPERS."717289");
END_REGION

REGION Network 14: CALL FB22503 HOPPER PRESSURE CONTROL HOPPER 1 UNIT 02
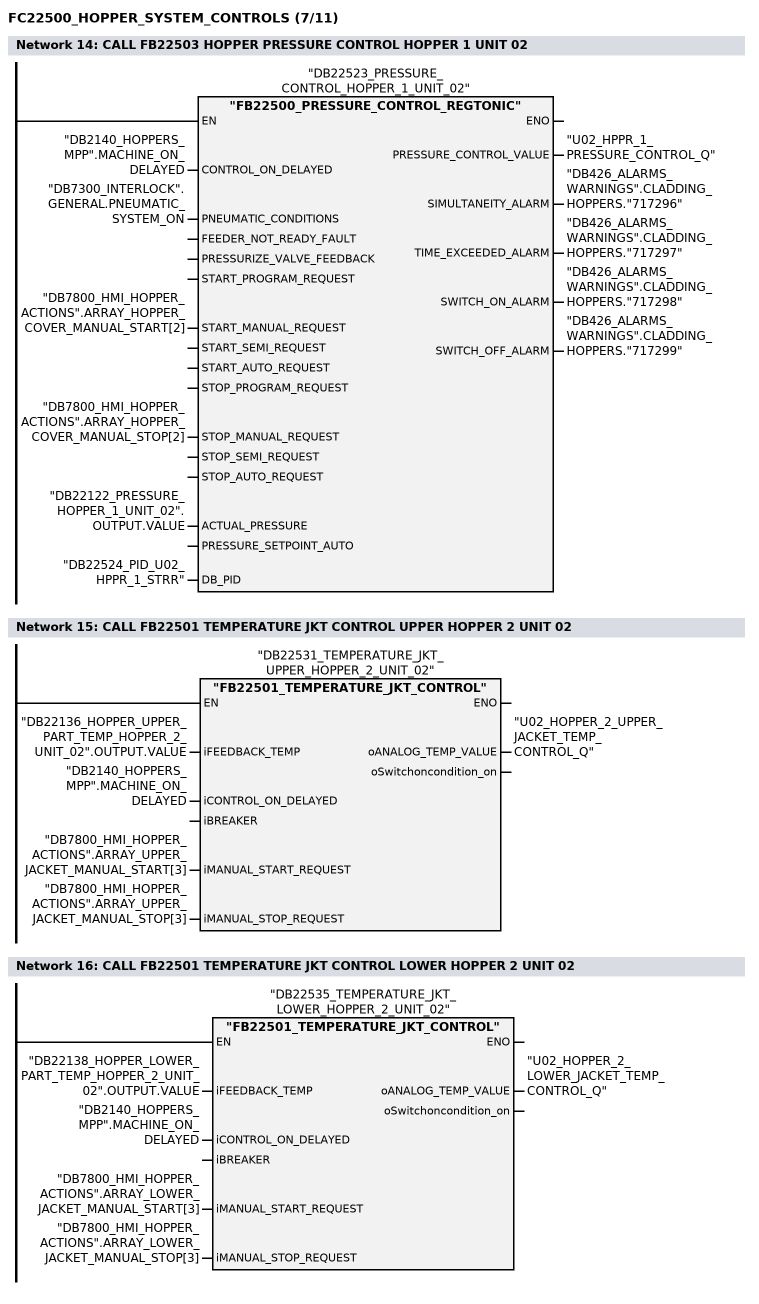
   RUNG wire#powerrail
      "DB22523_PRESSURE_CONTROL_HOPPER_1_UNIT_02"(CONTROL_ON_DELAYED := "DB2140_HOPPERS_MPP".MACHINE_ON_DELAYED, PNEUMATIC_CONDITIONS := "DB7300_INTERLOCK".GENERAL.PNEUMATIC_SYSTEM_ON, FEEDER_NOT_READY_FAULT :=, PRESSURIZE_VALVE_FEEDBACK :=, START_PROGRAM_REQUEST :=, START_MANUAL_REQUEST := "DB7800_HMI_HOPPER_ACTIONS".ARRAY_HOPPER_COVER_MANUAL_START[2], START_SEMI_REQUEST :=, START_AUTO_REQUEST :=, STOP_PROGRAM_REQUEST :=, STOP_MANUAL_REQUEST := "DB7800_HMI_HOPPER_ACTIONS".ARRAY_HOPPER_COVER_MANUAL_STOP[2], STOP_SEMI_REQUEST :=, STOP_AUTO_REQUEST :=, ACTUAL_PRESSURE := "DB22122_PRESSURE_HOPPER_1_UNIT_02".OUTPUT.VALUE, PRESSURE_SETPOINT_AUTO :=, DB_PID := "DB22524_PID_U02_HPPR_1_STRR", PRESSURE_CONTROL_VALUE => "U02_HPPR_1_PRESSURE_CONTROL_Q", SIMULTANEITY_ALARM => "DB426_ALARMS_WARNINGS".CLADDING_HOPPERS."717296", TIME_EXCEEDED_ALARM => "DB426_ALARMS_WARNINGS".CLADDING_HOPPERS."717297", SWITCH_ON_ALARM => "DB426_ALARMS_WARNINGS".CLADDING_HOPPERS."717298", SWITCH_OFF_ALARM => "DB426_ALARMS_WARNINGS".CLADDING_HOPPERS."717299")
   END_RUNG
   // the same network as SCL:
   "DB22523_PRESSURE_CONTROL_HOPPER_1_UNIT_02"(CONTROL_ON_DELAYED := "DB2140_HOPPERS_MPP".MACHINE_ON_DELAYED,   // "FB22500_PRESSURE_CONTROL_REGTONIC"
                           PNEUMATIC_CONDITIONS := "DB7300_INTERLOCK".GENERAL.PNEUMATIC_SYSTEM_ON,
                           START_MANUAL_REQUEST := "DB7800_HMI_HOPPER_ACTIONS".ARRAY_HOPPER_COVER_MANUAL_START[2],
                           STOP_MANUAL_REQUEST := "DB7800_HMI_HOPPER_ACTIONS".ARRAY_HOPPER_COVER_MANUAL_STOP[2],
                           ACTUAL_PRESSURE := "DB22122_PRESSURE_HOPPER_1_UNIT_02".OUTPUT.VALUE,
                           DB_PID := "DB22524_PID_U02_HPPR_1_STRR",
                           PRESSURE_CONTROL_VALUE => "U02_HPPR_1_PRESSURE_CONTROL_Q",
                           SIMULTANEITY_ALARM => "DB426_ALARMS_WARNINGS".CLADDING_HOPPERS."717296",
                           TIME_EXCEEDED_ALARM => "DB426_ALARMS_WARNINGS".CLADDING_HOPPERS."717297",
                           SWITCH_ON_ALARM => "DB426_ALARMS_WARNINGS".CLADDING_HOPPERS."717298",
                           SWITCH_OFF_ALARM => "DB426_ALARMS_WARNINGS".CLADDING_HOPPERS."717299");
END_REGION

REGION Network 15: CALL FB22501 TEMPERATURE JKT CONTROL UPPER HOPPER 2 UNIT 02
   RUNG wire#powerrail
      "DB22531_TEMPERATURE_JKT_UPPER_HOPPER_2_UNIT_02"(iFEEDBACK_TEMP := "DB22136_HOPPER_UPPER_PART_TEMP_HOPPER_2_UNIT_02".OUTPUT.VALUE, iCONTROL_ON_DELAYED := "DB2140_HOPPERS_MPP".MACHINE_ON_DELAYED, iBREAKER :=, iMANUAL_START_REQUEST := "DB7800_HMI_HOPPER_ACTIONS".ARRAY_UPPER_JACKET_MANUAL_START[3], iMANUAL_STOP_REQUEST := "DB7800_HMI_HOPPER_ACTIONS".ARRAY_UPPER_JACKET_MANUAL_STOP[3], oANALOG_TEMP_VALUE => "U02_HOPPER_2_UPPER_JACKET_TEMP_CONTROL_Q", oSwitchoncondition_on =>)
   END_RUNG
   // the same network as SCL:
   "DB22531_TEMPERATURE_JKT_UPPER_HOPPER_2_UNIT_02"(iFEEDBACK_TEMP := "DB22136_HOPPER_UPPER_PART_TEMP_HOPPER_2_UNIT_02".OUTPUT.VALUE,   // "FB22501_TEMPERATURE_JKT_CONTROL"
                           iCONTROL_ON_DELAYED := "DB2140_HOPPERS_MPP".MACHINE_ON_DELAYED,
                           iMANUAL_START_REQUEST := "DB7800_HMI_HOPPER_ACTIONS".ARRAY_UPPER_JACKET_MANUAL_START[3],
                           iMANUAL_STOP_REQUEST := "DB7800_HMI_HOPPER_ACTIONS".ARRAY_UPPER_JACKET_MANUAL_STOP[3],
                           oANALOG_TEMP_VALUE => "U02_HOPPER_2_UPPER_JACKET_TEMP_CONTROL_Q");
END_REGION

REGION Network 16: CALL FB22501 TEMPERATURE JKT CONTROL LOWER HOPPER 2 UNIT 02
   RUNG wire#powerrail
      "DB22535_TEMPERATURE_JKT_LOWER_HOPPER_2_UNIT_02"(iFEEDBACK_TEMP := "DB22138_HOPPER_LOWER_PART_TEMP_HOPPER_2_UNIT_02".OUTPUT.VALUE, iCONTROL_ON_DELAYED := "DB2140_HOPPERS_MPP".MACHINE_ON_DELAYED, iBREAKER :=, iMANUAL_START_REQUEST := "DB7800_HMI_HOPPER_ACTIONS".ARRAY_LOWER_JACKET_MANUAL_START[3], iMANUAL_STOP_REQUEST := "DB7800_HMI_HOPPER_ACTIONS".ARRAY_LOWER_JACKET_MANUAL_STOP[3], oANALOG_TEMP_VALUE => "U02_HOPPER_2_LOWER_JACKET_TEMP_CONTROL_Q", oSwitchoncondition_on =>)
   END_RUNG
   // the same network as SCL:
   "DB22535_TEMPERATURE_JKT_LOWER_HOPPER_2_UNIT_02"(iFEEDBACK_TEMP := "DB22138_HOPPER_LOWER_PART_TEMP_HOPPER_2_UNIT_02".OUTPUT.VALUE,   // "FB22501_TEMPERATURE_JKT_CONTROL"
                           iCONTROL_ON_DELAYED := "DB2140_HOPPERS_MPP".MACHINE_ON_DELAYED,
                           iMANUAL_START_REQUEST := "DB7800_HMI_HOPPER_ACTIONS".ARRAY_LOWER_JACKET_MANUAL_START[3],
                           iMANUAL_STOP_REQUEST := "DB7800_HMI_HOPPER_ACTIONS".ARRAY_LOWER_JACKET_MANUAL_STOP[3],
                           oANALOG_TEMP_VALUE => "U02_HOPPER_2_LOWER_JACKET_TEMP_CONTROL_Q");
END_REGION

REGION Network 17: CALL FB22502 MOTOR STIRRER CONTROL HOPPER 2 UNIT 02
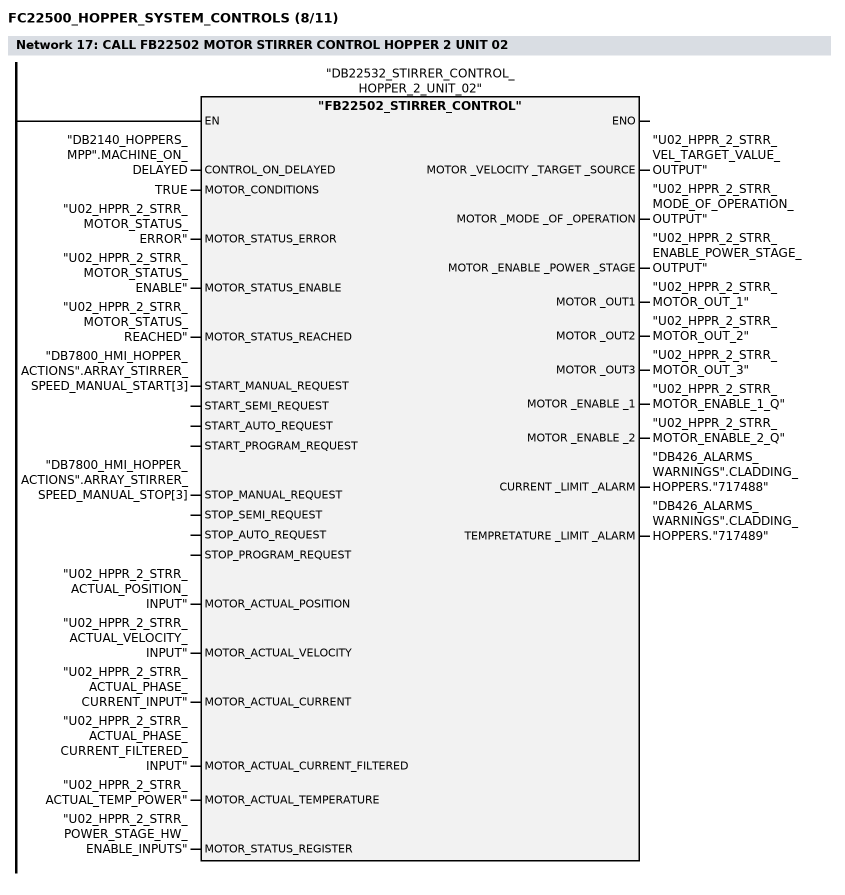
   RUNG wire#powerrail
      "DB22532_STIRRER_CONTROL_HOPPER_2_UNIT_02"(CONTROL_ON_DELAYED := "DB2140_HOPPERS_MPP".MACHINE_ON_DELAYED, MOTOR_CONDITIONS := TRUE, MOTOR_STATUS_ERROR := "U02_HPPR_2_STRR_MOTOR_STATUS_ERROR", MOTOR_STATUS_ENABLE := "U02_HPPR_2_STRR_MOTOR_STATUS_ENABLE", MOTOR_STATUS_REACHED := "U02_HPPR_2_STRR_MOTOR_STATUS_REACHED", START_MANUAL_REQUEST := "DB7800_HMI_HOPPER_ACTIONS".ARRAY_STIRRER_SPEED_MANUAL_START[3], START_SEMI_REQUEST :=, START_AUTO_REQUEST :=, START_PROGRAM_REQUEST :=, STOP_MANUAL_REQUEST := "DB7800_HMI_HOPPER_ACTIONS".ARRAY_STIRRER_SPEED_MANUAL_STOP[3], STOP_SEMI_REQUEST :=, STOP_AUTO_REQUEST :=, STOP_PROGRAM_REQUEST :=, MOTOR_ACTUAL_POSITION := "U02_HPPR_2_STRR_ACTUAL_POSITION_INPUT", MOTOR_ACTUAL_VELOCITY := "U02_HPPR_2_STRR_ACTUAL_VELOCITY_INPUT", MOTOR_ACTUAL_CURRENT := "U02_HPPR_2_STRR_ACTUAL_PHASE_CURRENT_INPUT", MOTOR_ACTUAL_CURRENT_FILTERED := "U02_HPPR_2_STRR_ACTUAL_PHASE_CURRENT_FILTERED_INPUT", MOTOR_ACTUAL_TEMPERATURE := "U02_HPPR_2_STRR_ACTUAL_TEMP_POWER", MOTOR_STATUS_REGISTER := "U02_HPPR_2_STRR_POWER_STAGE_HW_ENABLE_INPUTS", "MOTOR _VELOCITY _TARGET _SOURCE" => "U02_HPPR_2_STRR_VEL_TARGET_VALUE_OUTPUT", "MOTOR _MODE _OF _OPERATION" => "U02_HPPR_2_STRR_MODE_OF_OPERATION_OUTPUT", "MOTOR _ENABLE _POWER _STAGE" => "U02_HPPR_2_STRR_ENABLE_POWER_STAGE_OUTPUT", "MOTOR _OUT1" => "U02_HPPR_2_STRR_MOTOR_OUT_1", "MOTOR _OUT2" => "U02_HPPR_2_STRR_MOTOR_OUT_2", "MOTOR _OUT3" => "U02_HPPR_2_STRR_MOTOR_OUT_3", "MOTOR _ENABLE _1" => "U02_HPPR_2_STRR_MOTOR_ENABLE_1_Q", "MOTOR _ENABLE _2" => "U02_HPPR_2_STRR_MOTOR_ENABLE_2_Q", "CURRENT _LIMIT _ALARM" => "DB426_ALARMS_WARNINGS".CLADDING_HOPPERS."717488", "TEMPRETATURE _LIMIT _ALARM" => "DB426_ALARMS_WARNINGS".CLADDING_HOPPERS."717489")
   END_RUNG
   // the same network as SCL:
   "DB22532_STIRRER_CONTROL_HOPPER_2_UNIT_02"(CONTROL_ON_DELAYED := "DB2140_HOPPERS_MPP".MACHINE_ON_DELAYED,   // "FB22502_STIRRER_CONTROL"
                           MOTOR_CONDITIONS := TRUE,
                           MOTOR_STATUS_ERROR := "U02_HPPR_2_STRR_MOTOR_STATUS_ERROR",
                           MOTOR_STATUS_ENABLE := "U02_HPPR_2_STRR_MOTOR_STATUS_ENABLE",
                           MOTOR_STATUS_REACHED := "U02_HPPR_2_STRR_MOTOR_STATUS_REACHED",
                           START_MANUAL_REQUEST := "DB7800_HMI_HOPPER_ACTIONS".ARRAY_STIRRER_SPEED_MANUAL_START[3],
                           STOP_MANUAL_REQUEST := "DB7800_HMI_HOPPER_ACTIONS".ARRAY_STIRRER_SPEED_MANUAL_STOP[3],
                           MOTOR_ACTUAL_POSITION := "U02_HPPR_2_STRR_ACTUAL_POSITION_INPUT",
                           MOTOR_ACTUAL_VELOCITY := "U02_HPPR_2_STRR_ACTUAL_VELOCITY_INPUT",
                           MOTOR_ACTUAL_CURRENT := "U02_HPPR_2_STRR_ACTUAL_PHASE_CURRENT_INPUT",
                           MOTOR_ACTUAL_CURRENT_FILTERED := "U02_HPPR_2_STRR_ACTUAL_PHASE_CURRENT_FILTERED_INPUT",
                           MOTOR_ACTUAL_TEMPERATURE := "U02_HPPR_2_STRR_ACTUAL_TEMP_POWER",
                           MOTOR_STATUS_REGISTER := "U02_HPPR_2_STRR_POWER_STAGE_HW_ENABLE_INPUTS",
                           "MOTOR _VELOCITY _TARGET _SOURCE" => "U02_HPPR_2_STRR_VEL_TARGET_VALUE_OUTPUT",
                           "MOTOR _MODE _OF _OPERATION" => "U02_HPPR_2_STRR_MODE_OF_OPERATION_OUTPUT",
                           "MOTOR _ENABLE _POWER _STAGE" => "U02_HPPR_2_STRR_ENABLE_POWER_STAGE_OUTPUT",
                           "MOTOR _OUT1" => "U02_HPPR_2_STRR_MOTOR_OUT_1",
                           "MOTOR _OUT2" => "U02_HPPR_2_STRR_MOTOR_OUT_2",
                           "MOTOR _OUT3" => "U02_HPPR_2_STRR_MOTOR_OUT_3",
                           "MOTOR _ENABLE _1" => "U02_HPPR_2_STRR_MOTOR_ENABLE_1_Q",
                           "MOTOR _ENABLE _2" => "U02_HPPR_2_STRR_MOTOR_ENABLE_2_Q",
                           "CURRENT _LIMIT _ALARM" => "DB426_ALARMS_WARNINGS".CLADDING_HOPPERS."717488",
                           "TEMPRETATURE _LIMIT _ALARM" => "DB426_ALARMS_WARNINGS".CLADDING_HOPPERS."717489");
END_REGION

REGION Network 18: CALL FB22503 HOPPER PRESSURE CONTROL HOPPER 2 UNIT 02
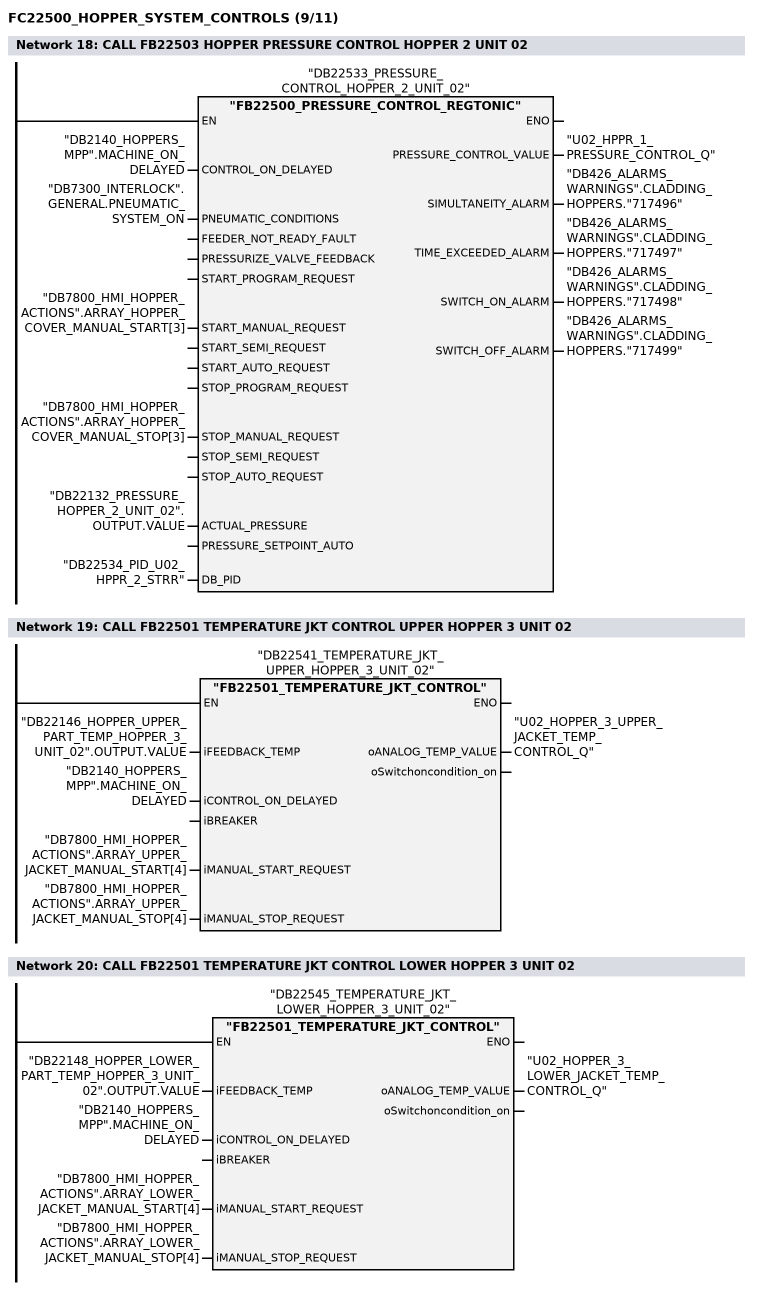
   RUNG wire#powerrail
      "DB22533_PRESSURE_CONTROL_HOPPER_2_UNIT_02"(CONTROL_ON_DELAYED := "DB2140_HOPPERS_MPP".MACHINE_ON_DELAYED, PNEUMATIC_CONDITIONS := "DB7300_INTERLOCK".GENERAL.PNEUMATIC_SYSTEM_ON, FEEDER_NOT_READY_FAULT :=, PRESSURIZE_VALVE_FEEDBACK :=, START_PROGRAM_REQUEST :=, START_MANUAL_REQUEST := "DB7800_HMI_HOPPER_ACTIONS".ARRAY_HOPPER_COVER_MANUAL_START[3], START_SEMI_REQUEST :=, START_AUTO_REQUEST :=, STOP_PROGRAM_REQUEST :=, STOP_MANUAL_REQUEST := "DB7800_HMI_HOPPER_ACTIONS".ARRAY_HOPPER_COVER_MANUAL_STOP[3], STOP_SEMI_REQUEST :=, STOP_AUTO_REQUEST :=, ACTUAL_PRESSURE := "DB22132_PRESSURE_HOPPER_2_UNIT_02".OUTPUT.VALUE, PRESSURE_SETPOINT_AUTO :=, DB_PID := "DB22534_PID_U02_HPPR_2_STRR", PRESSURE_CONTROL_VALUE => "U02_HPPR_1_PRESSURE_CONTROL_Q", SIMULTANEITY_ALARM => "DB426_ALARMS_WARNINGS".CLADDING_HOPPERS."717496", TIME_EXCEEDED_ALARM => "DB426_ALARMS_WARNINGS".CLADDING_HOPPERS."717497", SWITCH_ON_ALARM => "DB426_ALARMS_WARNINGS".CLADDING_HOPPERS."717498", SWITCH_OFF_ALARM => "DB426_ALARMS_WARNINGS".CLADDING_HOPPERS."717499")
   END_RUNG
   // the same network as SCL:
   "DB22533_PRESSURE_CONTROL_HOPPER_2_UNIT_02"(CONTROL_ON_DELAYED := "DB2140_HOPPERS_MPP".MACHINE_ON_DELAYED,   // "FB22500_PRESSURE_CONTROL_REGTONIC"
                           PNEUMATIC_CONDITIONS := "DB7300_INTERLOCK".GENERAL.PNEUMATIC_SYSTEM_ON,
                           START_MANUAL_REQUEST := "DB7800_HMI_HOPPER_ACTIONS".ARRAY_HOPPER_COVER_MANUAL_START[3],
                           STOP_MANUAL_REQUEST := "DB7800_HMI_HOPPER_ACTIONS".ARRAY_HOPPER_COVER_MANUAL_STOP[3],
                           ACTUAL_PRESSURE := "DB22132_PRESSURE_HOPPER_2_UNIT_02".OUTPUT.VALUE,
                           DB_PID := "DB22534_PID_U02_HPPR_2_STRR",
                           PRESSURE_CONTROL_VALUE => "U02_HPPR_1_PRESSURE_CONTROL_Q",
                           SIMULTANEITY_ALARM => "DB426_ALARMS_WARNINGS".CLADDING_HOPPERS."717496",
                           TIME_EXCEEDED_ALARM => "DB426_ALARMS_WARNINGS".CLADDING_HOPPERS."717497",
                           SWITCH_ON_ALARM => "DB426_ALARMS_WARNINGS".CLADDING_HOPPERS."717498",
                           SWITCH_OFF_ALARM => "DB426_ALARMS_WARNINGS".CLADDING_HOPPERS."717499");
END_REGION

REGION Network 19: CALL FB22501 TEMPERATURE JKT CONTROL UPPER HOPPER 3 UNIT 02
   RUNG wire#powerrail
      "DB22541_TEMPERATURE_JKT_UPPER_HOPPER_3_UNIT_02"(iFEEDBACK_TEMP := "DB22146_HOPPER_UPPER_PART_TEMP_HOPPER_3_UNIT_02".OUTPUT.VALUE, iCONTROL_ON_DELAYED := "DB2140_HOPPERS_MPP".MACHINE_ON_DELAYED, iBREAKER :=, iMANUAL_START_REQUEST := "DB7800_HMI_HOPPER_ACTIONS".ARRAY_UPPER_JACKET_MANUAL_START[4], iMANUAL_STOP_REQUEST := "DB7800_HMI_HOPPER_ACTIONS".ARRAY_UPPER_JACKET_MANUAL_STOP[4], oANALOG_TEMP_VALUE => "U02_HOPPER_3_UPPER_JACKET_TEMP_CONTROL_Q", oSwitchoncondition_on =>)
   END_RUNG
   // the same network as SCL:
   "DB22541_TEMPERATURE_JKT_UPPER_HOPPER_3_UNIT_02"(iFEEDBACK_TEMP := "DB22146_HOPPER_UPPER_PART_TEMP_HOPPER_3_UNIT_02".OUTPUT.VALUE,   // "FB22501_TEMPERATURE_JKT_CONTROL"
                           iCONTROL_ON_DELAYED := "DB2140_HOPPERS_MPP".MACHINE_ON_DELAYED,
                           iMANUAL_START_REQUEST := "DB7800_HMI_HOPPER_ACTIONS".ARRAY_UPPER_JACKET_MANUAL_START[4],
                           iMANUAL_STOP_REQUEST := "DB7800_HMI_HOPPER_ACTIONS".ARRAY_UPPER_JACKET_MANUAL_STOP[4],
                           oANALOG_TEMP_VALUE => "U02_HOPPER_3_UPPER_JACKET_TEMP_CONTROL_Q");
END_REGION

REGION Network 20: CALL FB22501 TEMPERATURE JKT CONTROL LOWER HOPPER 3 UNIT 02
   RUNG wire#powerrail
      "DB22545_TEMPERATURE_JKT_LOWER_HOPPER_3_UNIT_02"(iFEEDBACK_TEMP := "DB22148_HOPPER_LOWER_PART_TEMP_HOPPER_3_UNIT_02".OUTPUT.VALUE, iCONTROL_ON_DELAYED := "DB2140_HOPPERS_MPP".MACHINE_ON_DELAYED, iBREAKER :=, iMANUAL_START_REQUEST := "DB7800_HMI_HOPPER_ACTIONS".ARRAY_LOWER_JACKET_MANUAL_START[4], iMANUAL_STOP_REQUEST := "DB7800_HMI_HOPPER_ACTIONS".ARRAY_LOWER_JACKET_MANUAL_STOP[4], oANALOG_TEMP_VALUE => "U02_HOPPER_3_LOWER_JACKET_TEMP_CONTROL_Q", oSwitchoncondition_on =>)
   END_RUNG
   // the same network as SCL:
   "DB22545_TEMPERATURE_JKT_LOWER_HOPPER_3_UNIT_02"(iFEEDBACK_TEMP := "DB22148_HOPPER_LOWER_PART_TEMP_HOPPER_3_UNIT_02".OUTPUT.VALUE,   // "FB22501_TEMPERATURE_JKT_CONTROL"
                           iCONTROL_ON_DELAYED := "DB2140_HOPPERS_MPP".MACHINE_ON_DELAYED,
                           iMANUAL_START_REQUEST := "DB7800_HMI_HOPPER_ACTIONS".ARRAY_LOWER_JACKET_MANUAL_START[4],
                           iMANUAL_STOP_REQUEST := "DB7800_HMI_HOPPER_ACTIONS".ARRAY_LOWER_JACKET_MANUAL_STOP[4],
                           oANALOG_TEMP_VALUE => "U02_HOPPER_3_LOWER_JACKET_TEMP_CONTROL_Q");
END_REGION

REGION Network 21: CALL FB22502 MOTOR STIRRER CONTROL HOPPER 3 UNIT 02
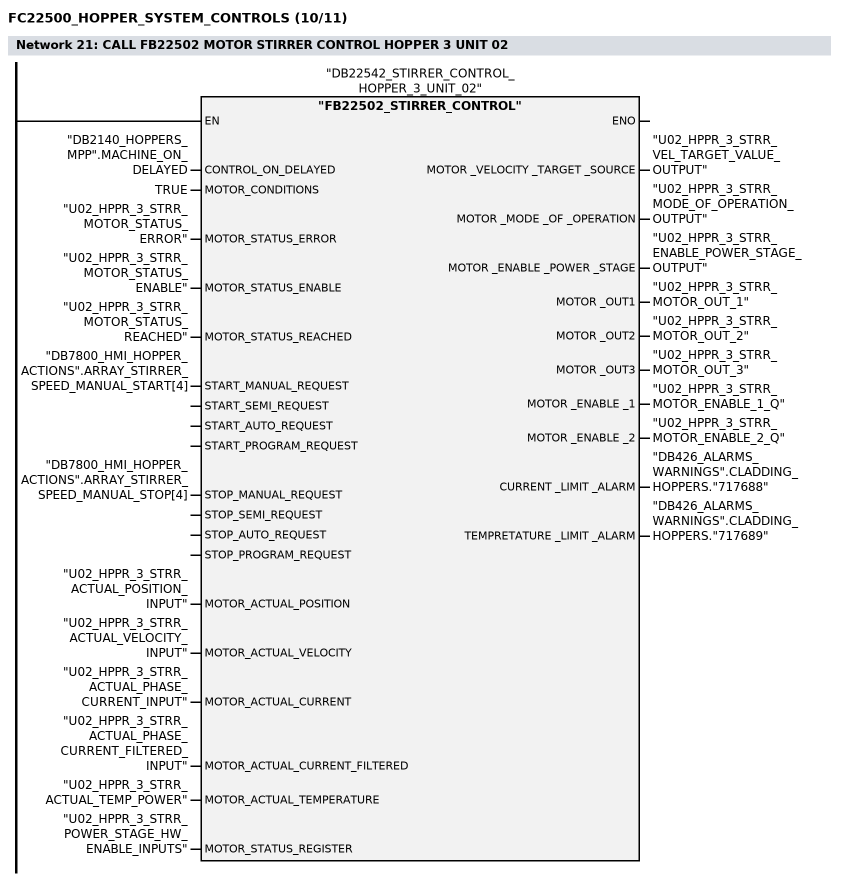
   RUNG wire#powerrail
      "DB22542_STIRRER_CONTROL_HOPPER_3_UNIT_02"(CONTROL_ON_DELAYED := "DB2140_HOPPERS_MPP".MACHINE_ON_DELAYED, MOTOR_CONDITIONS := TRUE, MOTOR_STATUS_ERROR := "U02_HPPR_3_STRR_MOTOR_STATUS_ERROR", MOTOR_STATUS_ENABLE := "U02_HPPR_3_STRR_MOTOR_STATUS_ENABLE", MOTOR_STATUS_REACHED := "U02_HPPR_3_STRR_MOTOR_STATUS_REACHED", START_MANUAL_REQUEST := "DB7800_HMI_HOPPER_ACTIONS".ARRAY_STIRRER_SPEED_MANUAL_START[4], START_SEMI_REQUEST :=, START_AUTO_REQUEST :=, START_PROGRAM_REQUEST :=, STOP_MANUAL_REQUEST := "DB7800_HMI_HOPPER_ACTIONS".ARRAY_STIRRER_SPEED_MANUAL_STOP[4], STOP_SEMI_REQUEST :=, STOP_AUTO_REQUEST :=, STOP_PROGRAM_REQUEST :=, MOTOR_ACTUAL_POSITION := "U02_HPPR_3_STRR_ACTUAL_POSITION_INPUT", MOTOR_ACTUAL_VELOCITY := "U02_HPPR_3_STRR_ACTUAL_VELOCITY_INPUT", MOTOR_ACTUAL_CURRENT := "U02_HPPR_3_STRR_ACTUAL_PHASE_CURRENT_INPUT", MOTOR_ACTUAL_CURRENT_FILTERED := "U02_HPPR_3_STRR_ACTUAL_PHASE_CURRENT_FILTERED_INPUT", MOTOR_ACTUAL_TEMPERATURE := "U02_HPPR_3_STRR_ACTUAL_TEMP_POWER", MOTOR_STATUS_REGISTER := "U02_HPPR_3_STRR_POWER_STAGE_HW_ENABLE_INPUTS", "MOTOR _VELOCITY _TARGET _SOURCE" => "U02_HPPR_3_STRR_VEL_TARGET_VALUE_OUTPUT", "MOTOR _MODE _OF _OPERATION" => "U02_HPPR_3_STRR_MODE_OF_OPERATION_OUTPUT", "MOTOR _ENABLE _POWER _STAGE" => "U02_HPPR_3_STRR_ENABLE_POWER_STAGE_OUTPUT", "MOTOR _OUT1" => "U02_HPPR_3_STRR_MOTOR_OUT_1", "MOTOR _OUT2" => "U02_HPPR_3_STRR_MOTOR_OUT_2", "MOTOR _OUT3" => "U02_HPPR_3_STRR_MOTOR_OUT_3", "MOTOR _ENABLE _1" => "U02_HPPR_3_STRR_MOTOR_ENABLE_1_Q", "MOTOR _ENABLE _2" => "U02_HPPR_3_STRR_MOTOR_ENABLE_2_Q", "CURRENT _LIMIT _ALARM" => "DB426_ALARMS_WARNINGS".CLADDING_HOPPERS."717688", "TEMPRETATURE _LIMIT _ALARM" => "DB426_ALARMS_WARNINGS".CLADDING_HOPPERS."717689")
   END_RUNG
   // the same network as SCL:
   "DB22542_STIRRER_CONTROL_HOPPER_3_UNIT_02"(CONTROL_ON_DELAYED := "DB2140_HOPPERS_MPP".MACHINE_ON_DELAYED,   // "FB22502_STIRRER_CONTROL"
                           MOTOR_CONDITIONS := TRUE,
                           MOTOR_STATUS_ERROR := "U02_HPPR_3_STRR_MOTOR_STATUS_ERROR",
                           MOTOR_STATUS_ENABLE := "U02_HPPR_3_STRR_MOTOR_STATUS_ENABLE",
                           MOTOR_STATUS_REACHED := "U02_HPPR_3_STRR_MOTOR_STATUS_REACHED",
                           START_MANUAL_REQUEST := "DB7800_HMI_HOPPER_ACTIONS".ARRAY_STIRRER_SPEED_MANUAL_START[4],
                           STOP_MANUAL_REQUEST := "DB7800_HMI_HOPPER_ACTIONS".ARRAY_STIRRER_SPEED_MANUAL_STOP[4],
                           MOTOR_ACTUAL_POSITION := "U02_HPPR_3_STRR_ACTUAL_POSITION_INPUT",
                           MOTOR_ACTUAL_VELOCITY := "U02_HPPR_3_STRR_ACTUAL_VELOCITY_INPUT",
                           MOTOR_ACTUAL_CURRENT := "U02_HPPR_3_STRR_ACTUAL_PHASE_CURRENT_INPUT",
                           MOTOR_ACTUAL_CURRENT_FILTERED := "U02_HPPR_3_STRR_ACTUAL_PHASE_CURRENT_FILTERED_INPUT",
                           MOTOR_ACTUAL_TEMPERATURE := "U02_HPPR_3_STRR_ACTUAL_TEMP_POWER",
                           MOTOR_STATUS_REGISTER := "U02_HPPR_3_STRR_POWER_STAGE_HW_ENABLE_INPUTS",
                           "MOTOR _VELOCITY _TARGET _SOURCE" => "U02_HPPR_3_STRR_VEL_TARGET_VALUE_OUTPUT",
                           "MOTOR _MODE _OF _OPERATION" => "U02_HPPR_3_STRR_MODE_OF_OPERATION_OUTPUT",
                           "MOTOR _ENABLE _POWER _STAGE" => "U02_HPPR_3_STRR_ENABLE_POWER_STAGE_OUTPUT",
                           "MOTOR _OUT1" => "U02_HPPR_3_STRR_MOTOR_OUT_1",
                           "MOTOR _OUT2" => "U02_HPPR_3_STRR_MOTOR_OUT_2",
                           "MOTOR _OUT3" => "U02_HPPR_3_STRR_MOTOR_OUT_3",
                           "MOTOR _ENABLE _1" => "U02_HPPR_3_STRR_MOTOR_ENABLE_1_Q",
                           "MOTOR _ENABLE _2" => "U02_HPPR_3_STRR_MOTOR_ENABLE_2_Q",
                           "CURRENT _LIMIT _ALARM" => "DB426_ALARMS_WARNINGS".CLADDING_HOPPERS."717688",
                           "TEMPRETATURE _LIMIT _ALARM" => "DB426_ALARMS_WARNINGS".CLADDING_HOPPERS."717689");
END_REGION

REGION Network 22: CALL FB22503 HOPPER PRESSURE CONTROL HOPPER 3 UNIT 02
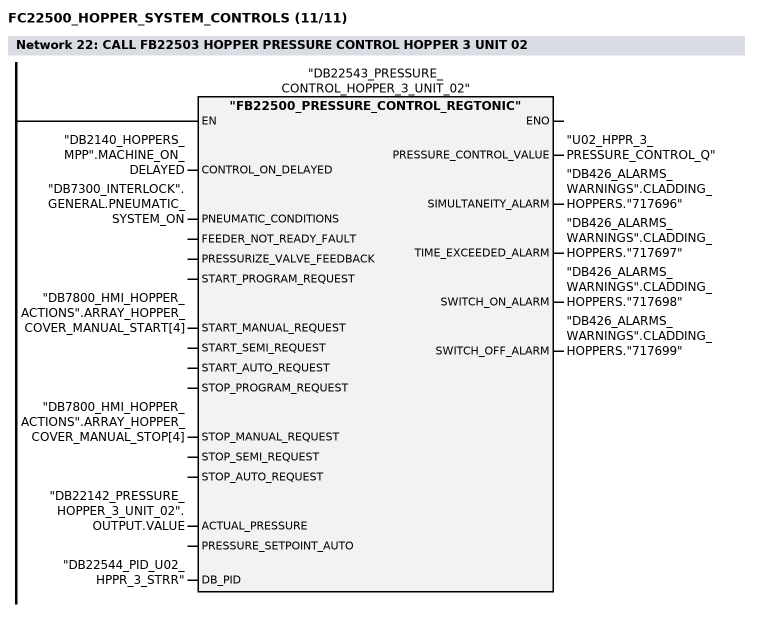
   RUNG wire#powerrail
      "DB22543_PRESSURE_CONTROL_HOPPER_3_UNIT_02"(CONTROL_ON_DELAYED := "DB2140_HOPPERS_MPP".MACHINE_ON_DELAYED, PNEUMATIC_CONDITIONS := "DB7300_INTERLOCK".GENERAL.PNEUMATIC_SYSTEM_ON, FEEDER_NOT_READY_FAULT :=, PRESSURIZE_VALVE_FEEDBACK :=, START_PROGRAM_REQUEST :=, START_MANUAL_REQUEST := "DB7800_HMI_HOPPER_ACTIONS".ARRAY_HOPPER_COVER_MANUAL_START[4], START_SEMI_REQUEST :=, START_AUTO_REQUEST :=, STOP_PROGRAM_REQUEST :=, STOP_MANUAL_REQUEST := "DB7800_HMI_HOPPER_ACTIONS".ARRAY_HOPPER_COVER_MANUAL_STOP[4], STOP_SEMI_REQUEST :=, STOP_AUTO_REQUEST :=, ACTUAL_PRESSURE := "DB22142_PRESSURE_HOPPER_3_UNIT_02".OUTPUT.VALUE, PRESSURE_SETPOINT_AUTO :=, DB_PID := "DB22544_PID_U02_HPPR_3_STRR", PRESSURE_CONTROL_VALUE => "U02_HPPR_3_PRESSURE_CONTROL_Q", SIMULTANEITY_ALARM => "DB426_ALARMS_WARNINGS".CLADDING_HOPPERS."717696", TIME_EXCEEDED_ALARM => "DB426_ALARMS_WARNINGS".CLADDING_HOPPERS."717697", SWITCH_ON_ALARM => "DB426_ALARMS_WARNINGS".CLADDING_HOPPERS."717698", SWITCH_OFF_ALARM => "DB426_ALARMS_WARNINGS".CLADDING_HOPPERS."717699")
   END_RUNG
   // the same network as SCL:
   "DB22543_PRESSURE_CONTROL_HOPPER_3_UNIT_02"(CONTROL_ON_DELAYED := "DB2140_HOPPERS_MPP".MACHINE_ON_DELAYED,   // "FB22500_PRESSURE_CONTROL_REGTONIC"
                           PNEUMATIC_CONDITIONS := "DB7300_INTERLOCK".GENERAL.PNEUMATIC_SYSTEM_ON,
                           START_MANUAL_REQUEST := "DB7800_HMI_HOPPER_ACTIONS".ARRAY_HOPPER_COVER_MANUAL_START[4],
                           STOP_MANUAL_REQUEST := "DB7800_HMI_HOPPER_ACTIONS".ARRAY_HOPPER_COVER_MANUAL_STOP[4],
                           ACTUAL_PRESSURE := "DB22142_PRESSURE_HOPPER_3_UNIT_02".OUTPUT.VALUE,
                           DB_PID := "DB22544_PID_U02_HPPR_3_STRR",
                           PRESSURE_CONTROL_VALUE => "U02_HPPR_3_PRESSURE_CONTROL_Q",
                           SIMULTANEITY_ALARM => "DB426_ALARMS_WARNINGS".CLADDING_HOPPERS."717696",
                           TIME_EXCEEDED_ALARM => "DB426_ALARMS_WARNINGS".CLADDING_HOPPERS."717697",
                           SWITCH_ON_ALARM => "DB426_ALARMS_WARNINGS".CLADDING_HOPPERS."717698",
                           SWITCH_OFF_ALARM => "DB426_ALARMS_WARNINGS".CLADDING_HOPPERS."717699");
END_REGION
END_FUNCTION
